// TwinCAT 3 PLC project TestPLC1
// ProgramVersion: 3.1.4023.0
// libraries:
//   Tc2_Standard, * (Beckhoff Automation GmbH)
//   Tc2_System, * (Beckhoff Automation GmbH)
//   Tc3_Module, * (Beckhoff Automation GmbH)
// project tree:
//   GVLs/ Grinder.TcGVL
//   / PlcTask.TcTTO
//   POUs/ MAIN.TcPOU, RunGrindingWell.TcPOU
// real-time tasks:
//   TASK PlcTask: cycle T#10ms, priority 20, ADS port 350

CONFIGURATION TestPLC1
    RESOURCE PLC ON TwinCAT3
        TASK PlcTask(INTERVAL := T#10ms, PRIORITY := 20);
        PROGRAM MAIN WITH PlcTask : MAIN;
    END_RESOURCE
END_CONFIGURATION

// ---- GVLs/Grinder.TcGVL
{attribute 'qualified_only'}
VAR_GLOBAL
	GridingWellMs AT %Q* : BOOL;
	StartGrindingWellPB AT %I* : BOOL;
	StopGrindingWellPB AT %I* : BOOL;
END_VAR

// ---- POUs/MAIN.TcPOU
PROGRAM MAIN
VAR
END_VAR

RunGrindingWell();

END_PROGRAM

// ---- POUs/RunGrindingWell.TcPOU
PROGRAM RunGrindingWell
VAR
END_VAR

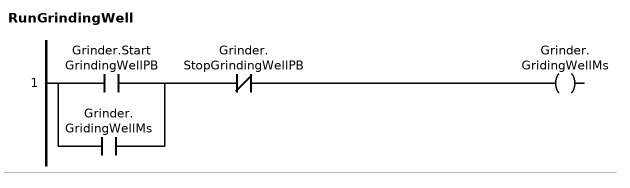
// NETWORK 1
Grinder.GridingWellMs := (Grinder.StartGrindingWellPB OR Grinder.GridingWellMs) AND NOT Grinder.StopGrindingWellPB;

END_PROGRAM
